FUNCTION_BLOCK PTRC_Protection_Trip_Conditioning (* Composite Function Block Type *)
  (* Standard: 61499-2 *)
  (* Version 0.0, 12/10/2023, Cheyan, Schneider Electric, template *)
  PACKAGE Main;
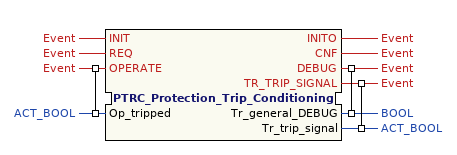
  EVENT_INPUT
    INIT; (* Initialization Request *)
    REQ; (* Normal Execution Request *)
    OPERATE WITH Op_tripped;
  END_EVENT
  EVENT_OUTPUT
    INITO; (* Initialization Confirm *)
    CNF; (* Execution Confirmation *)
    DEBUG WITH Tr_general_DEBUG;
    TR_TRIP_SIGNAL WITH Tr_trip_signal;
  END_EVENT
  VAR_INPUT
    Op_tripped : ACT_BOOL; (* Input event qualifier *)
  END_VAR
  VAR_OUTPUT
    Tr_general_DEBUG : BOOL;
    Tr_trip_signal : ACT_BOOL; (* Output event qualifier *)
  END_VAR
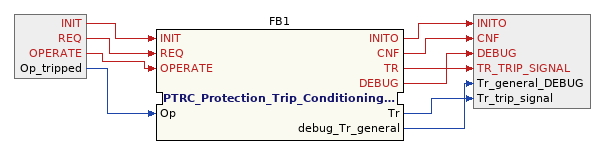
  FBS
    FB1 : PTRC_Protection_Trip_Conditioning_Logic;
  END_FBS
  EVENT_CONNECTIONS
    FB1.INITO TO INITO;
    FB1.CNF TO CNF;
    INIT TO FB1.INIT;
    REQ TO FB1.REQ;
    FB1.DEBUG TO DEBUG;
    OPERATE TO FB1.OPERATE;
    FB1.TR TO TR_TRIP_SIGNAL;
  END_CONNECTIONS
  DATA_CONNECTIONS
    FB1.debug_Tr_general TO Tr_general_DEBUG;
    Op_tripped TO FB1.Op;
    FB1.Tr TO Tr_trip_signal;
  END_CONNECTIONS
END_FUNCTION_BLOCK
